(* Logix 5000 project; controller VFX vendor 1 type 14 code 177 rev 31.11; software revision 31.00 *)

TASK LazyTask (periodic, rate 10 ms, priority 10, watchdog 500 ms) : Operator_Interface
TASK MainTask (continuous, watchdog 500 ms) : MainProgram, fanucProgram, VFX
TASK SafetyTask (periodic, rate 20 ms, priority 10, watchdog 20 ms, safety) : SafetyProgram

MODULES
   Local : vendor 1 type 14 code 177 (Compact 0, rev 31.11)
      IPC : ETHERNET-MODULE (Ethernet 192.168.1.253, rev 1.1, Output RPI 10 ms)
      TURCK_4AI : vendor 48 type 12 code 14025 (Ethernet 192.168.1.20, rev 2.7, StandardDataDriven RPI 20 ms)
      fanuc : vendor 356 type 140 code 40 (Ethernet 192.168.1.41, rev 3.1, StandardDataDriven RPI 32 ms, A_Safety_Output RPI 20 ms, B_Safety_Input RPI 10 ms)
      pointIO : 1734-AENTR (Ethernet 192.168.1.21, rev 5.1, Output RPI 20 ms)
         di8 : 1734-IB8 (PointIO 3, rev 3.1)
         ai2 : 1734-IE2V (PointIO 5, rev 3.1, Input RPI 80 ms)
         do8 : 1734-OB8 (PointIO 4, rev 3.1)
         si8 : vendor 1 type 35 code 15 (PointIO 1, rev 2.1, Input RPI 10 ms, Output RPI 20 ms)
         so8 : vendor 1 type 35 code 16 (PointIO 2, rev 2.1, Input RPI 10 ms, Output RPI 20 ms)
END_MODULES

TYPE BOXTYPE :
STRUCT
   name : STRING;
   fiducial1 : POSREG_T;
   fiducial2 : POSREG_T;
   slot00 : POSREG_T;
   rowpitch : DINT;
   colpitch : DINT;
   numrows : DINT;
   numcols : DINT;
END_STRUCT
END_TYPE

TYPE Buttons :
STRUCT
   Start : BOOL;
   Stop : BOOL;
   FaultReset : BOOL;
   EStopReset : BOOL;
   Request : BOOL;
END_STRUCT
END_TYPE

TYPE FANUC_DIN1_T :   // FANUC I/O Structure
STRUCT
   dw0 : FANUC_DWORDI10_T;
   dw1 : FANUC_DWORDI11_T;
   dw2 : FANUC_DWORDI12_T;
   dw3 : FANUC_DWORDI13_T;
END_STRUCT
END_TYPE

TYPE FANUC_DIO :
STRUCT
   camera_trigger_req : BOOL;
   gripper_hasItem : BOOL;
   tool_engage_req : BOOL;
   tool_release_req : BOOL;
   gripper_open_req : BOOL;
   gripper_close_req : BOOL;
   laser_trigger_req : BOOL;
   mode_AUTO : BOOL;
   mode_ESTOP : BOOL;
   mode_T1 : BOOL;
   camera_trigger_ACK : BOOL;
   gripper_isOpen : BOOL;
   laser_trigger_ACK : BOOL;
   tool_isEngaged : BOOL;
   toolnest1_isOpen : BOOL;
   toolnest2_isOpen : BOOL;
   toolnest3_isOpen : BOOL;
   light : SINT;
   gripper_isClosed : BOOL;
END_STRUCT
END_TYPE

TYPE FANUC_DOUT1_T :   // FANUC I/O Structure
STRUCT
   dw0 : FANUC_DWORDO10_T;
   dw1 : FANUC_DWORDO11_T;
   dw2 : FANUC_DWORDO12_T;
   dw3 : FANUC_DWORDO13_T;
END_STRUCT
END_TYPE

TYPE FANUC_DWORDI10_T :   // FANUC I/O Structure
STRUCT
   Wago_analog_input_1_DI1_GI1_1 : BOOL;
   Wago_analog_input_1_DI2_GI1_2 : BOOL;
   Wago_analog_input_1_DI3_GI1_4 : BOOL;
   Wago_analog_input_1_DI4_GI1_8 : BOOL;
   Wago_analog_input_1_DI5_GI1_16 : BOOL;
   Wago_analog_input_1_DI6_GI1_32 : BOOL;
   Wago_analog_input_1_DI7_GI1_64 : BOOL;
   Wago_analog_input_1_DI8_GI1_128 : BOOL;
   Wago_analog_input_1_DI9_GI1_1 : BOOL;
   Wago_analog_input_1_DI10_GI1_2 : BOOL;
   Wago_analog_input_1_DI11_GI1_4 : BOOL;
   Wago_analog_input_1_DI12_GI1_8 : BOOL;
   Wago_analog_input_1_DI13_GI1_16 : BOOL;
   Wago_analog_input_1_DI14_GI1_32 : BOOL;
   Wago_analog_input_1_DI15_GI1_64 : BOOL;
   Wago_analog_input_1_DI16_GI1_128 : BOOL;
   Wago_analog_input_2_DI17_GI2_1 : BOOL;
   Wago_analog_input_2_DI18_GI2_2 : BOOL;
   Wago_analog_input_2_DI19_GI2_4 : BOOL;
   Wago_analog_input_2_DI20_GI2_8 : BOOL;
   Wago_analog_input_2_DI21_GI2_16 : BOOL;
   Wago_analog_input_2_DI22_GI2_32 : BOOL;
   Wago_analog_input_2_DI23_GI2_64 : BOOL;
   Wago_analog_input_2_DI24_GI2_128 : BOOL;
   Wago_analog_input_2_DI25_GI2_1 : BOOL;
   Wago_analog_input_2_DI26_GI2_2 : BOOL;
   Wago_analog_input_2_DI27_GI2_4 : BOOL;
   Wago_analog_input_2_DI28_GI2_8 : BOOL;
   Wago_analog_input_2_DI29_GI2_16 : BOOL;
   Wago_analog_input_2_DI30_GI2_32 : BOOL;
   Wago_analog_input_2_DI31_GI2_64 : BOOL;
   Wago_analog_input_2_DI32_GI2_128 : BOOL;
END_STRUCT
END_TYPE

TYPE FANUC_DWORDI11_T :   // FANUC I/O Structure
STRUCT
   DI33 : BOOL;
   DI34 : BOOL;
   DI35 : BOOL;
   DI36 : BOOL;
   DI37 : BOOL;
   DI38 : BOOL;
   DI39 : BOOL;
   DI40 : BOOL;
   DI41 : BOOL;
   DI42 : BOOL;
   DI43 : BOOL;
   DI44 : BOOL;
   DI45 : BOOL;
   DI46 : BOOL;
   DI47 : BOOL;
   DI48 : BOOL;
   DI49 : BOOL;
   DI50 : BOOL;
   DI51 : BOOL;
   DI52 : BOOL;
   DI53 : BOOL;
   DI54 : BOOL;
   DI55 : BOOL;
   DI56 : BOOL;
   DI57 : BOOL;
   DI58 : BOOL;
   DI59 : BOOL;
   DI60 : BOOL;
   DI61 : BOOL;
   DI62 : BOOL;
   DI63 : BOOL;
   DI64 : BOOL;
END_STRUCT
END_TYPE

TYPE FANUC_DWORDI12_T :   // FANUC I/O Structure
STRUCT
   IMSTP_DI65_UI1 : BOOL;
   Hold_DI66_UI2 : BOOL;
   SFSPD_DI67_UI3 : BOOL;
   Cycle_stop_DI68_UI4 : BOOL;
   Fault_reset_DI69_UI5 : BOOL;
   Start_DI70_UI6 : BOOL;
   Home_DI71_UI7 : BOOL;
   Enable_DI72_UI8 : BOOL;
   RSR1PNS1STYLE1_DI73_UI9 : BOOL;
   RSR2PNS2STYLE2_DI74_UI10 : BOOL;
   RSR3PNS3STYLE3_DI75_UI11 : BOOL;
   RSR4PNS4STYLE4_DI76_UI12 : BOOL;
   RSR5PNS5STYLE5_DI77_UI13 : BOOL;
   RSR6PNS6STYLE6_DI78_UI14 : BOOL;
   RSR7PNS7STYLE7_DI79_UI15 : BOOL;
   RSR8PNS8STYLE8_DI80_UI16 : BOOL;
   PNS_strobe_DI81_UI17 : BOOL;
   Prod_start_DI82_UI18 : BOOL;
   DI83 : BOOL;
   DI84 : BOOL;
   DI85 : BOOL;
   DI86 : BOOL;
   DI87 : BOOL;
   DI88 : BOOL;
   DI89 : BOOL;
   DI90 : BOOL;
   DI91 : BOOL;
   DI92 : BOOL;
   DI93 : BOOL;
   DI94 : BOOL;
   DI95 : BOOL;
   DI96 : BOOL;
END_STRUCT
END_TYPE

TYPE FANUC_DWORDI13_T :   // FANUC I/O Structure
STRUCT
   DI97 : BOOL;
   DI98 : BOOL;
   DI99 : BOOL;
   Cognex_trig_ready_DI100 : BOOL;
   Cognex_trig_ack_DI101 : BOOL;
   Cognex_acquiring_DI102 : BOOL;
   Cognex_missed_ack_DI103 : BOOL;
   Cognex_online_DI104 : BOOL;
   Cognex_inspecting_DI105 : BOOL;
   Cognex_inspect_complete_DI106 : BOOL;
   Cognex_buffer_overrun_DI107 : BOOL;
   Cognex_results_valid_DI108 : BOOL;
   Cognex_job_loading_DI109 : BOOL;
   Cognex_job_load_complete_DI110 : BOOL;
   Cognex_job_load_failed_DI111 : BOOL;
   Cognex_exposure_complete_DI112 : BOOL;
   Cognex_job_pass_DI113 : BOOL;
   DI114 : BOOL;
   DI115 : BOOL;
   DI116 : BOOL;
   DI117 : BOOL;
   DI118 : BOOL;
   DI119 : BOOL;
   DI120 : BOOL;
   DI121 : BOOL;
   DI122 : BOOL;
   DI123 : BOOL;
   DI124 : BOOL;
   DI125 : BOOL;
   DI126 : BOOL;
   DI127 : BOOL;
   DI128 : BOOL;
END_STRUCT
END_TYPE

TYPE FANUC_DWORDO10_T :   // FANUC I/O Structure
STRUCT
   Camera_Trigger_DO1 : BOOL;
   Camera_Continouts_DO2 : BOOL;
   Laser_Trigger_DO3 : BOOL;
   Laser_Continous_DO4 : BOOL;
   DO5 : BOOL;
   DO6 : BOOL;
   DO7 : BOOL;
   DO8 : BOOL;
   DO9 : BOOL;
   DO10 : BOOL;
   DO11 : BOOL;
   DO12 : BOOL;
   DO13 : BOOL;
   DO14 : BOOL;
   DO15 : BOOL;
   DO16 : BOOL;
   DO17 : BOOL;
   DO18 : BOOL;
   DO19 : BOOL;
   DO20 : BOOL;
   DO21 : BOOL;
   DO22 : BOOL;
   DO23 : BOOL;
   DO24 : BOOL;
   DO25 : BOOL;
   DO26 : BOOL;
   DO27 : BOOL;
   DO28 : BOOL;
   DO29 : BOOL;
   DO30 : BOOL;
   DO31 : BOOL;
   DO32 : BOOL;
END_STRUCT
END_TYPE

TYPE FANUC_DWORDO11_T :   // FANUC I/O Structure
STRUCT
   DO33 : BOOL;
   DO34 : BOOL;
   DO35 : BOOL;
   DO36 : BOOL;
   DO37 : BOOL;
   DO38 : BOOL;
   DO39 : BOOL;
   DO40 : BOOL;
   DO41 : BOOL;
   DO42 : BOOL;
   DO43 : BOOL;
   DO44 : BOOL;
   DO45 : BOOL;
   DO46 : BOOL;
   DO47 : BOOL;
   DO48 : BOOL;
   DO49 : BOOL;
   DO50 : BOOL;
   DO51 : BOOL;
   DO52 : BOOL;
   DO53 : BOOL;
   DO54 : BOOL;
   DO55 : BOOL;
   DO56 : BOOL;
   DO57 : BOOL;
   DO58 : BOOL;
   DO59 : BOOL;
   DO60 : BOOL;
   DO61 : BOOL;
   DO62 : BOOL;
   DO63 : BOOL;
   DO64 : BOOL;
END_STRUCT
END_TYPE

TYPE FANUC_DWORDO12_T :   // FANUC I/O Structure
STRUCT
   Cmd_enabled_DO65_UO1 : BOOL;
   System_ready_DO66_UO2 : BOOL;
   Prg_running_DO67_UO3 : BOOL;
   Prg_paused_DO68_UO4 : BOOL;
   Motion_held_DO69_UO5 : BOOL;
   Fault_DO70_UO6 : BOOL;
   At_perch_DO71_UO7 : BOOL;
   TP_enabled_DO72_UO8 : BOOL;
   Batt_alarm_DO73_UO9 : BOOL;
   Busy_DO74_UO10 : BOOL;
   ACK1SNO1_DO75_UO11 : BOOL;
   ACK2SNO2_DO76_UO12 : BOOL;
   ACK3SNO3_DO77_UO13 : BOOL;
   ACK4SNO4_DO78_UO14 : BOOL;
   ACK5SNO5_DO79_UO15 : BOOL;
   ACK6SNO6_DO80_UO16 : BOOL;
   ACK7SNO7_DO81_UO17 : BOOL;
   ACK8SNO8_DO82_UO18 : BOOL;
   SNACK_DO83_UO19 : BOOL;
   Reserved_DO84_UO20 : BOOL;
   DO85 : BOOL;
   DO86 : BOOL;
   DO87 : BOOL;
   DO88 : BOOL;
   DO89 : BOOL;
   DO90 : BOOL;
   DO91 : BOOL;
   DO92 : BOOL;
   DO93 : BOOL;
   DO94 : BOOL;
   DO95 : BOOL;
   DO96 : BOOL;
END_STRUCT
END_TYPE

TYPE FANUC_DWORDO13_T :   // FANUC I/O Structure
STRUCT
   DO97 : BOOL;
   DO98 : BOOL;
   DO99 : BOOL;
   Cognex_trigger_enable_DO100 : BOOL;
   Cognex_trigger_DO101 : BOOL;
   Cognex_buffer_results_en_DO102 : BOOL;
   Cognex_inspect_result_ok_DO103 : BOOL;
   Cognex_reserved_DO104 : BOOL;
   Cognex_reserved_DO105 : BOOL;
   Cognex_reserved_DO106 : BOOL;
   Cognex_set_offline_DO107 : BOOL;
   Cognex_soft_event_0_DO108 : BOOL;
   Cognex_soft_event_1_DO109 : BOOL;
   Cognex_soft_event_2_DO110 : BOOL;
   Cognex_soft_event_3_DO111 : BOOL;
   Cognex_soft_event_4_DO112 : BOOL;
   Cognex_soft_event_5_DO113 : BOOL;
   Cognex_soft_event_6_DO114 : BOOL;
   Cognex_soft_event_7_DO115 : BOOL;
   Cognex_reserved_DO116 : BOOL;
   Cognex_reserved_DO117 : BOOL;
   Cognex_reserved_DO118 : BOOL;
   Cognex_reserved_DO119 : BOOL;
   Cognex_reserved_DO120 : BOOL;
   Cognex_reserved_DO121 : BOOL;
   Cognex_reserved_DO122 : BOOL;
   Cognex_reserved_DO123 : BOOL;
   Cognex_reserved_DO124 : BOOL;
   Cognex_reserved_DO125 : BOOL;
   Cognex_reserved_DO126 : BOOL;
   Cognex_reserved_DO127 : BOOL;
   Cognex_reserved_DO128 : BOOL;
END_STRUCT
END_TYPE

TYPE FANUC_EDA_T :
STRUCT
   out : FANUC_I_T;
   in : FANUC_O_T;
END_STRUCT
END_TYPE

TYPE FANUC_I_T :
STRUCT
   dout : FANUC_DIN1_T;
   speed_max_R1 : DINT;
   speed_camera_R2 : DINT;
   speed_laser_R3 : DINT;
   speed_approach_R4 : DINT;
   R5 : DINT;
   R6 : DINT;
   R7 : DINT;
   R8 : DINT;
   speedj_max_R9 : DINT;
   speedj_payload_R10 : DINT;
   boxtype_numrows_R11 : DINT;
   boxtype_numcols_R12 : DINT;
   camera_getmode_R13 : DINT;
   laser_distance_R14 : DINT;
   camera_getfiducl_R15 : DINT;
   skip_perch_R16 : DINT;
   R17 : DINT;
   boxtype_ID_R18 : DINT;
   boxtype_rowpitch_R19 : DINT;
   boxtype_colpitch_R20 : DINT;
   target_boxnum_R21 : DINT;
   target_slotrow_R22 : DINT;
   target_slotcol_R23 : DINT;
   R24 : DINT;
   boxtype_fid1_PR1_G1 : POSREG_T;
   boxtype_fid2_PR2_G1 : POSREG_T;
   boxtype_slot00_PR3_G1 : POSREG_T;
   boxframe_offset_PR4_G1 : POSREG_T;
END_STRUCT
END_TYPE

TYPE FANUC_MASTER :
STRUCT
   uop : FANUC_UOPS;
   reg : FANUC_REGISTERS;
   dio : FANUC_DIO;
END_STRUCT
END_TYPE

TYPE FANUC_O_T :
STRUCT
   din : FANUC_DOUT1_T;
   speed_max_R1 : DINT;
   speed_camera_R2 : DINT;
   speed_laser_R3 : DINT;
   speed_approach_R4 : DINT;
   R5 : DINT;
   R6 : DINT;
   R7 : DINT;
   R8 : DINT;
   speedj_max_R9 : DINT;
   speedj_payload_R10 : DINT;
   boxtype_numrows_R11 : DINT;
   boxtype_numcols_R12 : DINT;
   camera_getmode_R13 : DINT;
   laser_distance_R14 : DINT;
   camera_getfiducl_R15 : DINT;
   skip_perch_R16 : DINT;
   R17 : DINT;
   boxtype_ID_R18 : DINT;
   boxtype_rowpitch_R19 : DINT;
   boxtype_colpitch_R20 : DINT;
   target_boxnum_R21 : DINT;
   target_slotrow_R22 : DINT;
   target_slotcol_R23 : DINT;
   R24 : DINT;
   R25 : DINT;
   R26 : DINT;
   R27 : DINT;
   R28 : DINT;
   R29 : DINT;
   R30 : DINT;
   style_result_R31 : DINT;
   row_current_R32 : DINT;
   boxtype_fid1_PR1_G1 : POSREG_T;
   boxtype_fid2_PR2_G1 : POSREG_T;
   boxtype_slot00_PR3_G1 : POSREG_T;
   boxframe_offset_PR4_G1 : POSREG_T;
   eda1_PR5_G1 : POSREG_T;
   eda2_PR6_G1 : POSREG_T;
   CURPOS_G1 : POSREG_T;
END_STRUCT
END_TYPE

TYPE FANUC_REGISTERS :
STRUCT
   boxframe_offset : POSREG_T;
   boxframe_offset_ACK : POSREG_T;
   boxtype : BOXTYPE;
   boxtype_ACK : BOXTYPE;
   laser_distance : DINT;
   speed_approach : DINT;
   speed_max : DINT;
   speed_payload : DINT;
   speed_toolchange : DINT;
   target_boxnum : DINT;
   target_slotrow : DINT;
   target_slotcol : DINT;
   target_tool_ID : DINT;
   CURPOS : POSREG_T;
   EDA1 : POSREG_T;
   EDA2 : POSREG_T;
   laser_distance_ACK : DINT;
   speed_approach_ACK : DINT;
   speed_max_ACK : DINT;
   speed_payload_ACK : DINT;
   speed_toolchange_ACK : DINT;
   speedj_max_ACK : DINT;
   speedJ_payload_ACK : DINT;
   target_boxnum_ACK : DINT;
   target_slotrow_ACK : DINT;
   target_slotcol_ACK : DINT;
   current_tool_ID : DINT;
   target_fiducial : DINT;
   target_fiducial_ACK : DINT;
   style_result : DINT;
END_STRUCT
END_TYPE

TYPE FANUC_UOPS :
STRUCT
   cycle_stop : BOOL;
   enable : BOOL;
   fault_reset : BOOL;
   hold : BOOL;
   home : BOOL;
   IMSTP : BOOL;
   pns_strobe : BOOL;
   prod_start : BOOL;
   style : SINT;
   SFSPD : BOOL;
   start : BOOL;
   style_ACK : SINT;
   at_perch : BOOL;
   batt_alarm : BOOL;
   busy : BOOL;
   cmd_enabled : BOOL;
   fault : BOOL;
   motion_held : BOOL;
   prg_paused : BOOL;
   prg_running : BOOL;
   reserved : BOOL;
   SNACK : BOOL;
   system_ready : BOOL;
   TP_enabled : BOOL;
END_STRUCT
END_TYPE

TYPE Pedestal_Lights :
STRUCT
   Start : BOOL;
   Stop : BOOL;
   FaultReset : BOOL;
   EStopReset : BOOL;
   Request : BOOL;
   EStop : BOOL;
   White : BOOL;
   Blue : BOOL;
   Green : BOOL;
   Amber : BOOL;
   Red : BOOL;
   White_Flasher : BOOL;
   Blue_Flasher : BOOL;
   Green_Flasher : BOOL;
   Amber_Flasher : BOOL;
   Red_Flasher : BOOL;
END_STRUCT
END_TYPE

TYPE POSREG_T :   // FANUC Position Register (Cartesian Mode)
STRUCT
   uframe : INT;
   utool : INT;
   X : REAL;
   Y : REAL;
   Z : REAL;
   W : REAL;
   P : REAL;
   R : REAL;
   turn1 : SINT;
   turn2 : SINT;
   turn3 : SINT;
   front : BOOL;
   up : BOOL;
   left : BOOL;
   flip : BOOL;
   ext : REAL[3];
END_STRUCT
END_TYPE

VAR_GLOBAL   (* controller tags *)
   boxtypes : BOXTYPE[10] := ([0].name := 'tote', [0].fiducial1.uframe := -1, [0].fiducial1.front := 1, [0].fiducial1.up := 1, [0].fiducial1.left := 1, [0].fiducial2.uframe := -1, [0].fiducial2.X := 580.0, [0].fiducial2.Z := -220.0, [0].fiducial2.front := 1, [0].fiducial2.up := 1, [0].fiducial2.left := 1, [0].slot00.uframe := -1, [0].slot00.X := 60.0, [0].slot00.Y := 60.0, [0].slot00.Z := -295.0, [0].slot00.front := 1, [0].slot00.up := 1, [0].slot00.left := 1, [0].rowpitch := 42164, [0].colpitch := 128016, [0].numrows := 12, [0].numcols := 2, [1].name := 'carton1', [1].fiducial1.uframe := 63, [1].fiducial1.utool := 31, [1].fiducial1.X := 100.0, [1].fiducial1.Y := 40.0, [1].fiducial1.front := 1, [1].fiducial1.up := 1, [1].fiducial1.left := 1, [1].fiducial2.uframe := 63, [1].fiducial2.utool := 31, [1].fiducial2.X := 377.0, [1].fiducial2.Z := -220.0, [1].fiducial2.front := 1, [1].fiducial2.up := 1, [1].fiducial2.left := 1, [1].slot00.uframe := -1, [1].slot00.X := -18.5, [1].slot00.Y := 60.0, [1].slot00.Z := -295.0, [1].slot00.front := 1, [1].slot00.up := 1, [1].slot00.left := 1, [1].rowpitch := 47350, [1].colpitch := 122428, [1].numrows := 10, [1].numcols := 2);
   fanuc : FANUC_MASTER := (uop.enable := 1, uop.hold := 1, uop.IMSTP := 1, uop.style := 3, uop.SFSPD := 1, uop.cmd_enabled := 1, reg.boxframe_offset.uframe := -1, reg.boxframe_offset.X := 11.01, reg.boxframe_offset.Y := -9.029, reg.boxtype.name := 'tote', reg.boxtype.fiducial1.uframe := -1, reg.boxtype.fiducial1.front := 1, reg.boxtype.fiducial1.up := 1, reg.boxtype.fiducial1.left := 1, reg.boxtype.fiducial2.uframe := -1, reg.boxtype.fiducial2.X := 580.0, reg.boxtype.fiducial2.Z := -220.0, reg.boxtype.fiducial2.front := 1, reg.boxtype.fiducial2.up := 1, reg.boxtype.fiducial2.left := 1, reg.boxtype.slot00.uframe := -1, reg.boxtype.slot00.X := 60.0, reg.boxtype.slot00.Y := 60.0, reg.boxtype.slot00.Z := -295.0, reg.boxtype.slot00.front := 1, reg.boxtype.slot00.up := 1, reg.boxtype.slot00.left := 1, reg.boxtype.rowpitch := 42164, reg.boxtype.colpitch := 128016, reg.boxtype.numrows := 12, reg.boxtype.numcols := 2, reg.speed_approach := 1000, reg.speed_max := 2000, reg.speed_payload := 2000, reg.speed_toolchange := 2000, reg.target_boxnum := 7, reg.target_slotrow := 11, reg.target_slotcol := 1, reg.CURPOS.uframe := 7, reg.CURPOS.utool := 1, reg.CURPOS.X := 523.80383, reg.CURPOS.Y := -68.01611, reg.CURPOS.Z := -294.99994, reg.CURPOS.W := -1.6060338e-05, reg.CURPOS.P := 0.00042976913, reg.CURPOS.R := 1.6143189e-05, reg.CURPOS.front := 1, reg.CURPOS.up := 1, reg.EDA1.uframe := 255, reg.EDA1.utool := 255, reg.EDA1.X := nan, reg.EDA1.Y := nan, reg.EDA1.Z := nan, reg.EDA1.W := nan, reg.EDA1.P := nan, reg.EDA1.R := nan, reg.style_result := 1);
   fanuc_auto_enable : BOOL := 1;
   Fanuc_AUTO_OFF : BOOL := 1;
   Fanuc_ESTOP : EMERGENCY_STOP := (ChannelA := 1, ChannelB := 1, CircuitReset := 1, FaultReset := 1, O1 := 1);
   Fanuc_ESTOP_IN : BOOL := 1;
   Fanuc_ESTOP_OUT : BOOL := 1;
   Fanuc_FENCE : BOOL := 1;
   fanuc_IPC_start : BOOL;
   fanuc_permissive : BOOL := 1;
   fanuc_run : BOOL := 1;
   fanuc_s1 : FANUC_EDA_T := (out.dout.dw2.IMSTP_DI65_UI1 := 1, out.dout.dw2.Hold_DI66_UI2 := 1, out.dout.dw2.SFSPD_DI67_UI3 := 1, out.dout.dw2.Enable_DI72_UI8 := 1, out.dout.dw2.RSR1PNS1STYLE1_DI73_UI9 := 1, out.dout.dw2.RSR2PNS2STYLE2_DI74_UI10 := 1, out.speed_max_R1 := 2000, out.speed_camera_R2 := 2000, out.speed_laser_R3 := 1000, out.speed_approach_R4 := 2000, out.speedj_max_R9 := 100, out.speedj_payload_R10 := 100, out.boxtype_numrows_R11 := 12, out.boxtype_numcols_R12 := 2, out.boxtype_rowpitch_R19 := 42164, out.boxtype_colpitch_R20 := 128016, out.target_boxnum_R21 := 7, out.target_slotrow_R22 := 11, out.target_slotcol_R23 := 1, out.boxtype_fid1_PR1_G1.uframe := -1, out.boxtype_fid1_PR1_G1.front := 1, out.boxtype_fid1_PR1_G1.up := 1, out.boxtype_fid1_PR1_G1.left := 1, out.boxtype_fid2_PR2_G1.uframe := -1, out.boxtype_fid2_PR2_G1.X := 580.0, out.boxtype_fid2_PR2_G1.Z := -220.0, out.boxtype_fid2_PR2_G1.front := 1, out.boxtype_fid2_PR2_G1.up := 1, out.boxtype_fid2_PR2_G1.left := 1, out.boxtype_slot00_PR3_G1.uframe := -1, out.boxtype_slot00_PR3_G1.X := 60.0, out.boxtype_slot00_PR3_G1.Y := 60.0, out.boxtype_slot00_PR3_G1.Z := -295.0, out.boxtype_slot00_PR3_G1.front := 1, out.boxtype_slot00_PR3_G1.up := 1, out.boxtype_slot00_PR3_G1.left := 1, out.boxframe_offset_PR4_G1.uframe := -1, out.boxframe_offset_PR4_G1.X := 11.01, out.boxframe_offset_PR4_G1.Y := -9.029, in.din.dw2.Cmd_enabled_DO65_UO1 := 1, in.din.dw2.System_ready_DO66_UO2 := 1, in.speed_max_R1 := 2000, in.speed_camera_R2 := 2000, in.speed_laser_R3 := 1000, in.speed_approach_R4 := 2000, in.speedj_max_R9 := 100, in.speedj_payload_R10 := 100, in.boxtype_numrows_R11 := 12, in.boxtype_numcols_R12 := 2, in.boxtype_rowpitch_R19 := 42164, in.boxtype_colpitch_R20 := 128016, in.target_boxnum_R21 := 7, in.target_slotrow_R22 := 11, in.target_slotcol_R23 := 1, in.style_result_R31 := 1, in.boxtype_fid1_PR1_G1.uframe := 255, in.boxtype_fid1_PR1_G1.utool := 255, in.boxtype_fid1_PR1_G1.front := 1, in.boxtype_fid1_PR1_G1.up := 1, in.boxtype_fid1_PR1_G1.left := 1,
        in.boxtype_fid2_PR2_G1.uframe := 255, in.boxtype_fid2_PR2_G1.utool := 255, in.boxtype_fid2_PR2_G1.X := 580.0, in.boxtype_fid2_PR2_G1.Z := -220.0, in.boxtype_fid2_PR2_G1.front := 1, in.boxtype_fid2_PR2_G1.up := 1, in.boxtype_fid2_PR2_G1.left := 1, in.boxtype_slot00_PR3_G1.uframe := 255, in.boxtype_slot00_PR3_G1.utool := 255, in.boxtype_slot00_PR3_G1.X := 60.0, in.boxtype_slot00_PR3_G1.Y := 60.0, in.boxtype_slot00_PR3_G1.Z := -295.0, in.boxtype_slot00_PR3_G1.front := 1, in.boxtype_slot00_PR3_G1.up := 1, in.boxtype_slot00_PR3_G1.left := 1, in.boxframe_offset_PR4_G1.uframe := 255, in.boxframe_offset_PR4_G1.utool := 255, in.boxframe_offset_PR4_G1.X := 11.01, in.boxframe_offset_PR4_G1.Y := -9.029, in.eda1_PR5_G1.uframe := 255, in.eda1_PR5_G1.utool := 255, in.eda1_PR5_G1.X := nan, in.eda1_PR5_G1.Y := nan, in.eda1_PR5_G1.Z := nan, in.eda1_PR5_G1.W := nan, in.eda1_PR5_G1.P := nan, in.eda1_PR5_G1.R := nan, in.eda2_PR6_G1.uframe := 255, in.eda2_PR6_G1.utool := 255, in.eda2_PR6_G1.X := nan, in.eda2_PR6_G1.Y := nan, in.eda2_PR6_G1.Z := nan, in.eda2_PR6_G1.W := nan, in.eda2_PR6_G1.P := nan, in.eda2_PR6_G1.R := nan, in.CURPOS_G1.uframe := 7, in.CURPOS_G1.utool := 1, in.CURPOS_G1.X := 523.80383, in.CURPOS_G1.Y := -68.01611, in.CURPOS_G1.Z := -294.99994, in.CURPOS_G1.W := -1.6060338e-05, in.CURPOS_G1.P := 0.00042976913, in.CURPOS_G1.R := 1.6143189e-05, in.CURPOS_G1.front := 1, in.CURPOS_G1.up := 1);
   fanuc_style_start : BOOL;
   fanuc_target_boxtype : DINT;
   fanuc_target_valid : BOOL := 1;
   FENCE_CLOSED : BOOL := 1;
   HMI_Buttons : Buttons;
   HMI_Buttons2 : BOOL;
   HMI_ESTOP_Reset : BOOL;
   light_flasher : TIMER := (PRE := 500, ACC := 500, EN := 1, DN := 1);
   light_flasher2 : TIMER := (PRE := 500, ACC := 220, EN := 1, TT := 1);
   out_fail2 : BOOL := 1;
   out_pass2 : BOOL;
   output_pulse2 : DINT := 250;
   Panel_HMI_Lights : Pedestal_Lights;
   Panel_Stack_Amber : BOOL;
   Panel_Stack_Amber_Flasher : BOOL;
   Panel_Stack_Green : BOOL;
   Panel_Stack_Green_Flasher : BOOL := 1;
   Panel_Stack_Red : BOOL;
   Panel_Stack_Red_Flasher : BOOL;
   Pedestal1_ESTOP : EMERGENCY_STOP := (ResetType := 1, ChannelA := 1, ChannelB := 1, CircuitReset := 1, O1 := 1);
   Pedestal2_ESTOP : EMERGENCY_STOP := (ResetType := 1, ChannelA := 1, ChannelB := 1, CircuitReset := 1, O1 := 1);
   Safety_EStopReset : BOOL := 1;
   Safety_FaultReset : BOOL := 1;
   shhhhhhhhhh : BOOL;
   step_robot_command : DINT := 40;
   System_ESTOP : BOOL := 1;
   System_EStopReset : BOOL := 1;
   System_EStopResetReq : BOOL;
   System_FaultReset2 : BOOL;
   system_running : BOOL;
   system_running_debounce : TIMER := (PRE := 500, ACC := 500);
   System_Start : BOOL;
   System_Start2 : BOOL;
   System_Stop : BOOL;
   System_Stop2 : BOOL;
   tmr_pulse_fanuc : TIMER := (PRE := 500);
   tmr_pulse_fanuc_done : TIMER := (PRE := 500);
   tmr_start_fanuc : TIMER := (PRE := 100);
   vfx_laser_distance : INT[2];
END_VAR

PROGRAM fanucProgram   (* main routine fanucRoutine *)

ROUTINE fanucRoutine   (* ladder *)
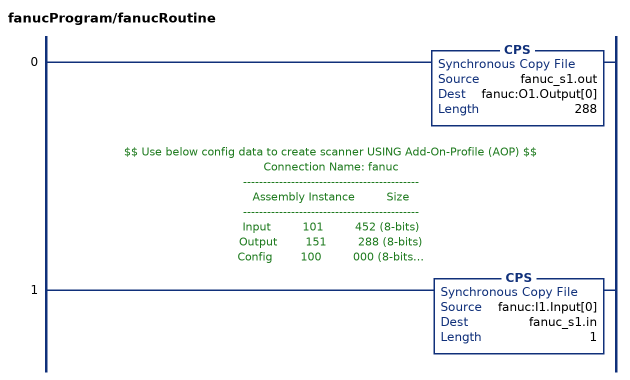
   0: CPS(fanuc_s1.out,fanuc:O1.Output[0],288);
   // $$ Use below config data to create scanner USING Add-On-Profile (AOP) $$
   //                   Connection Name: fanuc
   //                 --------------------------------------------
   //                   Assembly Instance         Size
   //                 --------------------------------------------
   //                   Input         101         452 (8-bits)
   //                   Output        151         288 (8-bits)
   //                   Config        100         000 (8-bits)
   //                 --------------------------------------------
   1: CPS(fanuc:I1.Input[0],fanuc_s1.in,1);
END_ROUTINE
END_PROGRAM

PROGRAM MainProgram   (* main routine MainRoutine *)

ROUTINE MainRoutine   (* ladder *)
   0 (stored rung type 13): ;
END_ROUTINE
END_PROGRAM

PROGRAM Operator_Interface   (* main routine Main_OI *)

ROUTINE Buttons_IO   (* ladder *)
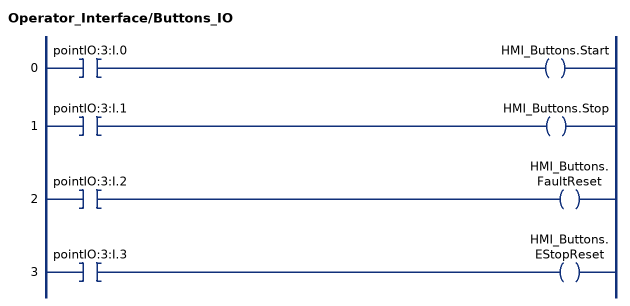
   0: XIC(pointIO:3:I.0)OTE(HMI_Buttons.Start);
   1: XIC(pointIO:3:I.1)OTE(HMI_Buttons.Stop);
   2: XIC(pointIO:3:I.2)OTE(HMI_Buttons.FaultReset);
   3: XIC(pointIO:3:I.3)OTE(HMI_Buttons.EStopReset);
END_ROUTINE

ROUTINE Buttons_Logic   (* ladder *)
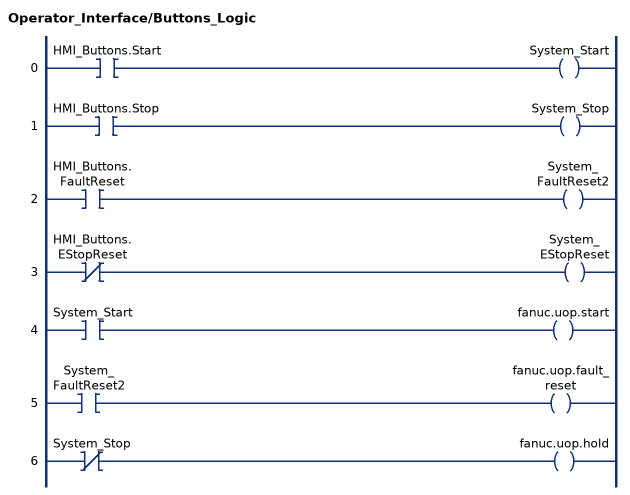
   0: XIC(HMI_Buttons.Start)OTE(System_Start);
   1: XIC(HMI_Buttons.Stop)OTE(System_Stop);
   2: XIC(HMI_Buttons.FaultReset)OTE(System_FaultReset2);
   3: XIO(HMI_Buttons.EStopReset)OTE(System_EStopReset);
   4: XIC(System_Start)OTE(fanuc.uop.start);
   5: XIC(System_FaultReset2)OTE(fanuc.uop.fault_reset);
   6: XIO(System_Stop)OTE(fanuc.uop.hold);
END_ROUTINE

ROUTINE Lights_IO   (* ladder *)
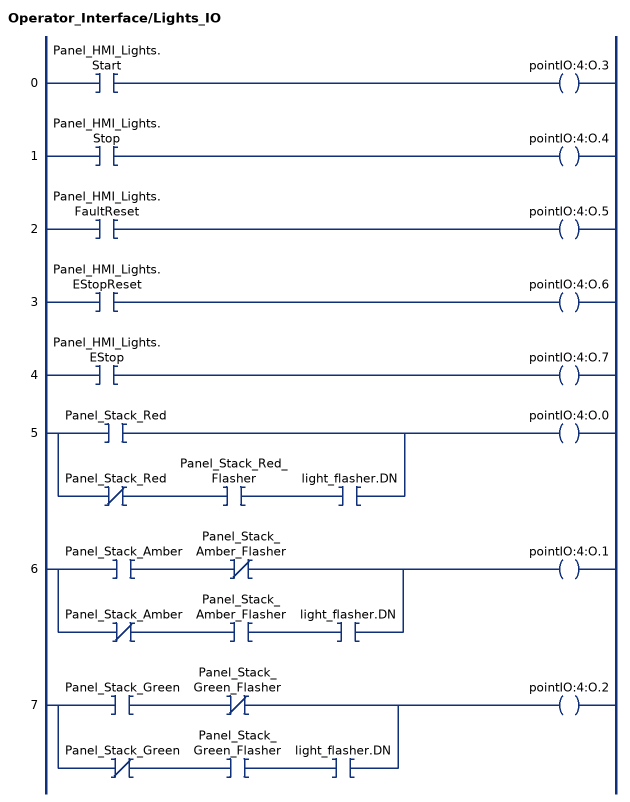
   0: XIC(Panel_HMI_Lights.Start)OTE(pointIO:4:O.3);
   1: XIC(Panel_HMI_Lights.Stop)OTE(pointIO:4:O.4);
   2: XIC(Panel_HMI_Lights.FaultReset)OTE(pointIO:4:O.5);
   3: XIC(Panel_HMI_Lights.EStopReset)OTE(pointIO:4:O.6);
   4: XIC(Panel_HMI_Lights.EStop)OTE(pointIO:4:O.7);
   5: [XIC(Panel_Stack_Red) ,XIO(Panel_Stack_Red) XIC(Panel_Stack_Red_Flasher) XIC(light_flasher.DN) ]OTE(pointIO:4:O.0);
   6: [XIC(Panel_Stack_Amber) XIO(Panel_Stack_Amber_Flasher) ,XIO(Panel_Stack_Amber) XIC(Panel_Stack_Amber_Flasher) XIC(light_flasher.DN) ]OTE(pointIO:4:O.1);
   7: [XIC(Panel_Stack_Green) XIO(Panel_Stack_Green_Flasher) ,XIO(Panel_Stack_Green) XIC(Panel_Stack_Green_Flasher) XIC(light_flasher.DN) ]OTE(pointIO:4:O.2);
END_ROUTINE

ROUTINE Lights_Logic   (* ladder *)
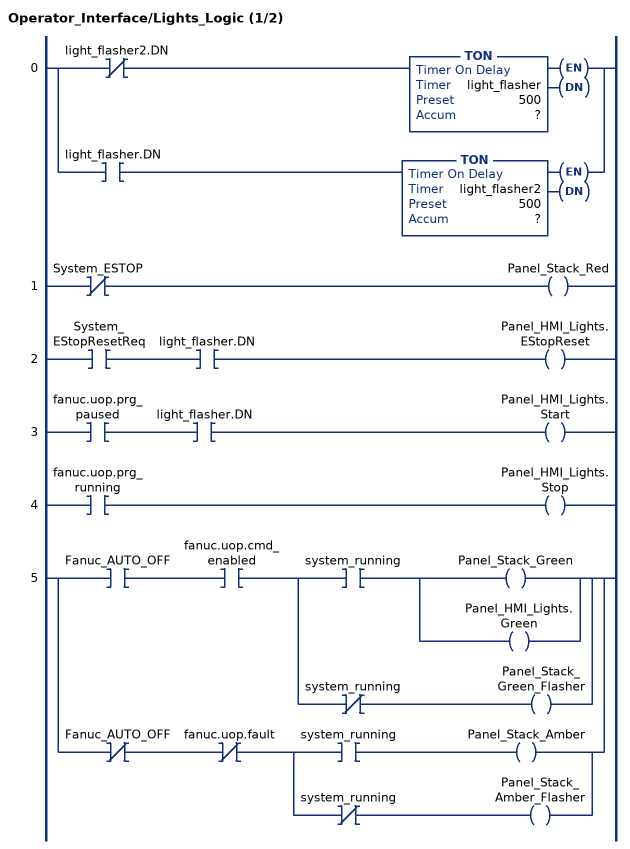
   0: [XIO(light_flasher2.DN) TON(light_flasher,?,?) ,XIC(light_flasher.DN) TON(light_flasher2,?,?) ];
   1: XIO(System_ESTOP)OTE(Panel_Stack_Red);
   2: XIC(System_EStopResetReq)XIC(light_flasher.DN)OTE(Panel_HMI_Lights.EStopReset);
   3: XIC(fanuc.uop.prg_paused)XIC(light_flasher.DN)OTE(Panel_HMI_Lights.Start);
   4: XIC(fanuc.uop.prg_running)OTE(Panel_HMI_Lights.Stop);
   5: [XIC(Fanuc_AUTO_OFF) XIC(fanuc.uop.cmd_enabled) [XIC(system_running) [OTE(Panel_Stack_Green) ,OTE(Panel_HMI_Lights.Green) ] ,XIO(system_running) OTE(Panel_Stack_Green_Flasher) ] ,XIO(Fanuc_AUTO_OFF) XIO(fanuc.uop.fault) [XIC(system_running) OTE(Panel_Stack_Amber) ,XIO(system_running) OTE(Panel_Stack_Amber_Flasher) ] ];
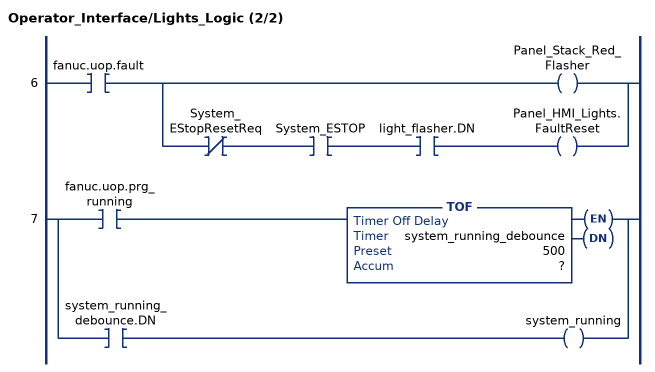
   6: XIC(fanuc.uop.fault)[OTE(Panel_Stack_Red_Flasher) ,XIO(System_EStopResetReq) XIC(System_ESTOP) XIC(light_flasher.DN) OTE(Panel_HMI_Lights.FaultReset) ];
   7: [XIC(fanuc.uop.prg_running) TOF(system_running_debounce,?,?) ,XIC(system_running_debounce.DN) OTE(system_running) ];
END_ROUTINE

ROUTINE Main_OI   (* ladder *)
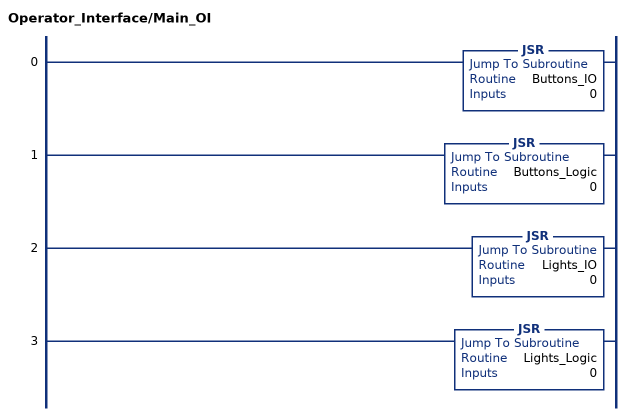
   0: JSR(Buttons_IO,0);
   1: JSR(Buttons_Logic,0);
   2: JSR(Lights_IO,0);
   3: JSR(Lights_Logic,0);
END_ROUTINE
END_PROGRAM

PROGRAM SafetyProgram   (* main routine MainRoutine, safety *)

ROUTINE ESTOPS   (* ladder *)
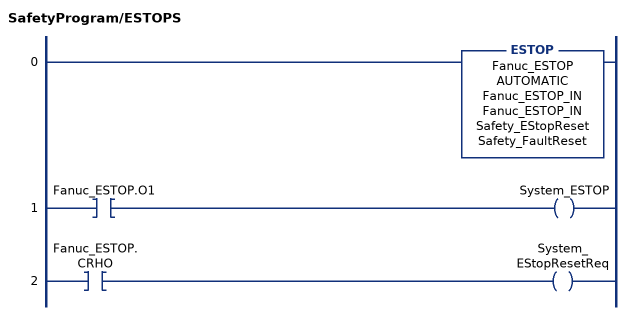
   0: ESTOP(Fanuc_ESTOP,AUTOMATIC,Fanuc_ESTOP_IN,Fanuc_ESTOP_IN,Safety_EStopReset,Safety_FaultReset);
   1: XIC(Fanuc_ESTOP.O1)OTE(System_ESTOP);
   2: XIC(Fanuc_ESTOP.CRHO)OTE(System_EStopResetReq);
END_ROUTINE

ROUTINE IO_Map   (* ladder *)
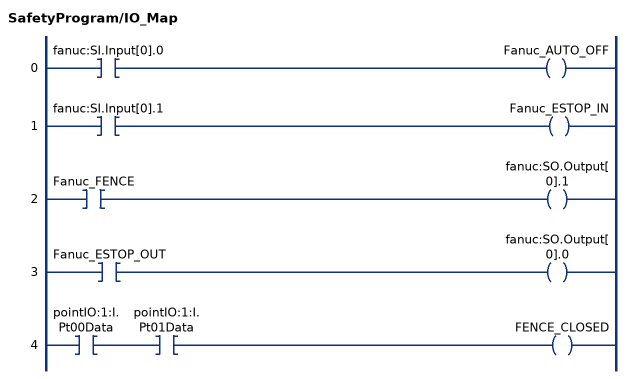
   0: XIC(fanuc:SI.Input[0].0)OTE(Fanuc_AUTO_OFF);
   1: XIC(fanuc:SI.Input[0].1)OTE(Fanuc_ESTOP_IN);
   2: XIC(Fanuc_FENCE)OTE(fanuc:SO.Output[0].1);
   3: XIC(Fanuc_ESTOP_OUT)OTE(fanuc:SO.Output[0].0);
   4: XIC(pointIO:1:I.Pt00Data)XIC(pointIO:1:I.Pt01Data)OTE(FENCE_CLOSED);
END_ROUTINE

ROUTINE MainRoutine   (* ladder *)
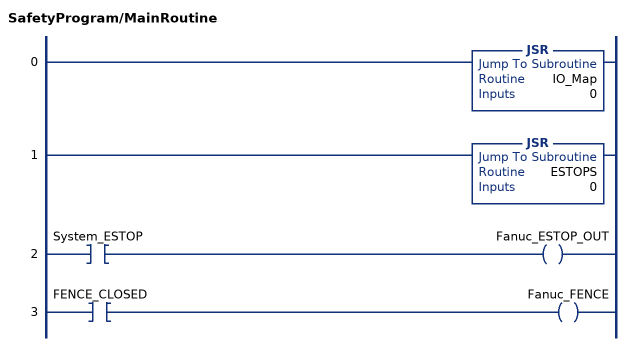
   0: JSR(IO_Map,0);
   1: JSR(ESTOPS,0);
   2: XIC(System_ESTOP)OTE(Fanuc_ESTOP_OUT);
   3: XIC(FENCE_CLOSED)OTE(Fanuc_FENCE);
END_ROUTINE
END_PROGRAM

PROGRAM VFX   (* main routine MainRoutine *)

ROUTINE Demo3   (* ladder *)
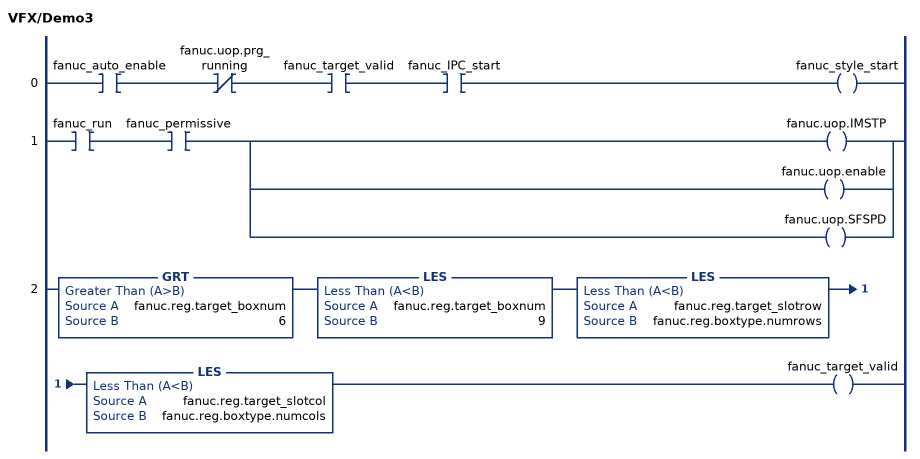
   0: XIC(fanuc_auto_enable)XIO(fanuc.uop.prg_running)XIC(fanuc_target_valid)XIC(fanuc_IPC_start)OTE(fanuc_style_start);
   1: XIC(fanuc_run)XIC(fanuc_permissive)[OTE(fanuc.uop.IMSTP) ,OTE(fanuc.uop.enable) ,OTE(fanuc.uop.SFSPD) ];
   2: GRT(fanuc.reg.target_boxnum,6)LES(fanuc.reg.target_boxnum,9)LES(fanuc.reg.target_slotrow,fanuc.reg.boxtype.numrows)LES(fanuc.reg.target_slotcol,fanuc.reg.boxtype.numcols)OTE(fanuc_target_valid);
END_ROUTINE

ROUTINE fanuc_IO   (* ladder *)
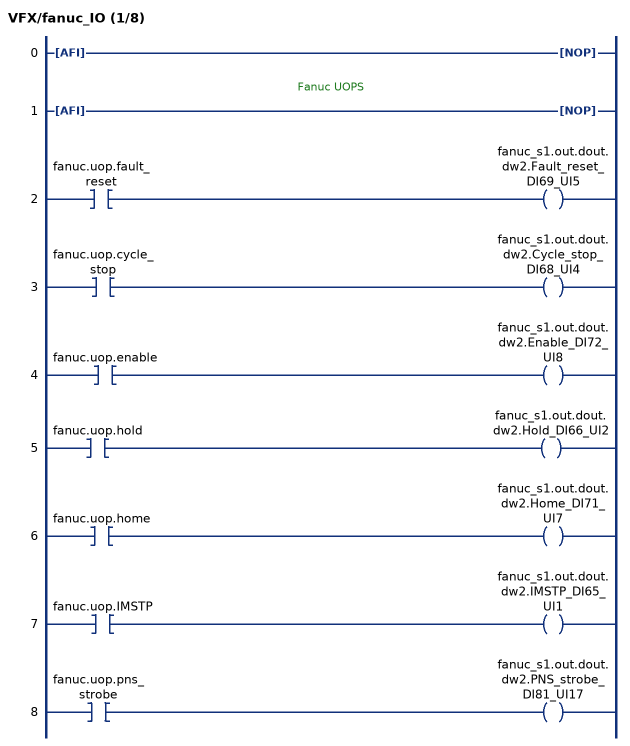
   0: AFI()NOP();
   // Fanuc UOPS
   1: AFI()NOP();
   2: XIC(fanuc.uop.fault_reset)OTE(fanuc_s1.out.dout.dw2.Fault_reset_DI69_UI5);
   3: XIC(fanuc.uop.cycle_stop)OTE(fanuc_s1.out.dout.dw2.Cycle_stop_DI68_UI4);
   4: XIC(fanuc.uop.enable)OTE(fanuc_s1.out.dout.dw2.Enable_DI72_UI8);
   5: XIC(fanuc.uop.hold)OTE(fanuc_s1.out.dout.dw2.Hold_DI66_UI2);
   6: XIC(fanuc.uop.home)OTE(fanuc_s1.out.dout.dw2.Home_DI71_UI7);
   7: XIC(fanuc.uop.IMSTP)OTE(fanuc_s1.out.dout.dw2.IMSTP_DI65_UI1);
   8: XIC(fanuc.uop.pns_strobe)OTE(fanuc_s1.out.dout.dw2.PNS_strobe_DI81_UI17);
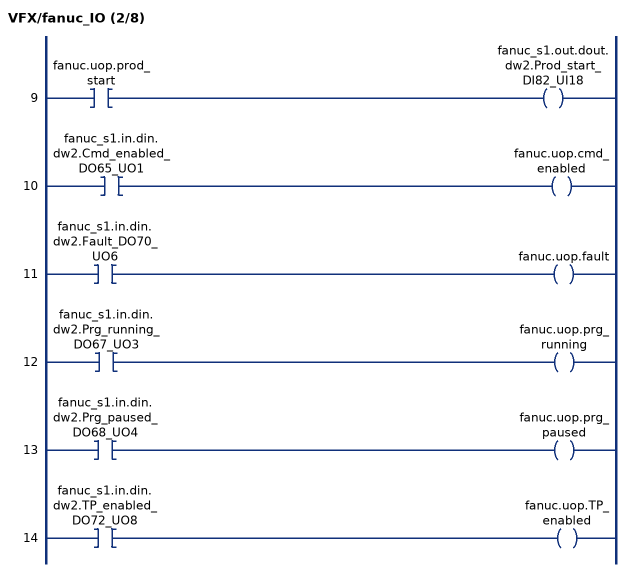
   9: XIC(fanuc.uop.prod_start)OTE(fanuc_s1.out.dout.dw2.Prod_start_DI82_UI18);
   10: XIC(fanuc_s1.in.din.dw2.Cmd_enabled_DO65_UO1)OTE(fanuc.uop.cmd_enabled);
   11: XIC(fanuc_s1.in.din.dw2.Fault_DO70_UO6)OTE(fanuc.uop.fault);
   12: XIC(fanuc_s1.in.din.dw2.Prg_running_DO67_UO3)OTE(fanuc.uop.prg_running);
   13: XIC(fanuc_s1.in.din.dw2.Prg_paused_DO68_UO4)OTE(fanuc.uop.prg_paused);
   14: XIC(fanuc_s1.in.din.dw2.TP_enabled_DO72_UO8)OTE(fanuc.uop.TP_enabled);
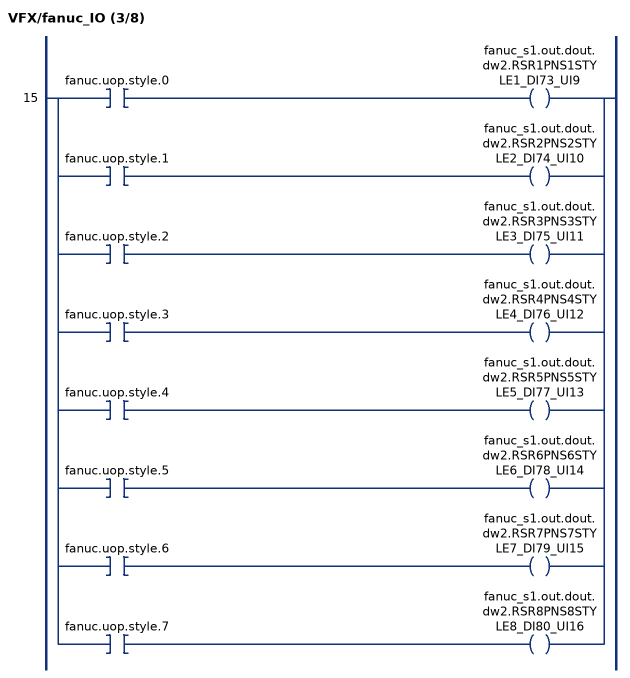
   15: [XIC(fanuc.uop.style.0) OTE(fanuc_s1.out.dout.dw2.RSR1PNS1STYLE1_DI73_UI9) ,XIC(fanuc.uop.style.1) OTE(fanuc_s1.out.dout.dw2.RSR2PNS2STYLE2_DI74_UI10) ,XIC(fanuc.uop.style.2) OTE(fanuc_s1.out.dout.dw2.RSR3PNS3STYLE3_DI75_UI11) ,XIC(fanuc.uop.style.3) OTE(fanuc_s1.out.dout.dw2.RSR4PNS4STYLE4_DI76_UI12) ,XIC(fanuc.uop.style.4) OTE(fanuc_s1.out.dout.dw2.RSR5PNS5STYLE5_DI77_UI13) ,XIC(fanuc.uop.style.5) OTE(fanuc_s1.out.dout.dw2.RSR6PNS6STYLE6_DI78_UI14) ,XIC(fanuc.uop.style.6) OTE(fanuc_s1.out.dout.dw2.RSR7PNS7STYLE7_DI79_UI15) ,XIC(fanuc.uop.style.7) OTE(fanuc_s1.out.dout.dw2.RSR8PNS8STYLE8_DI80_UI16) ];
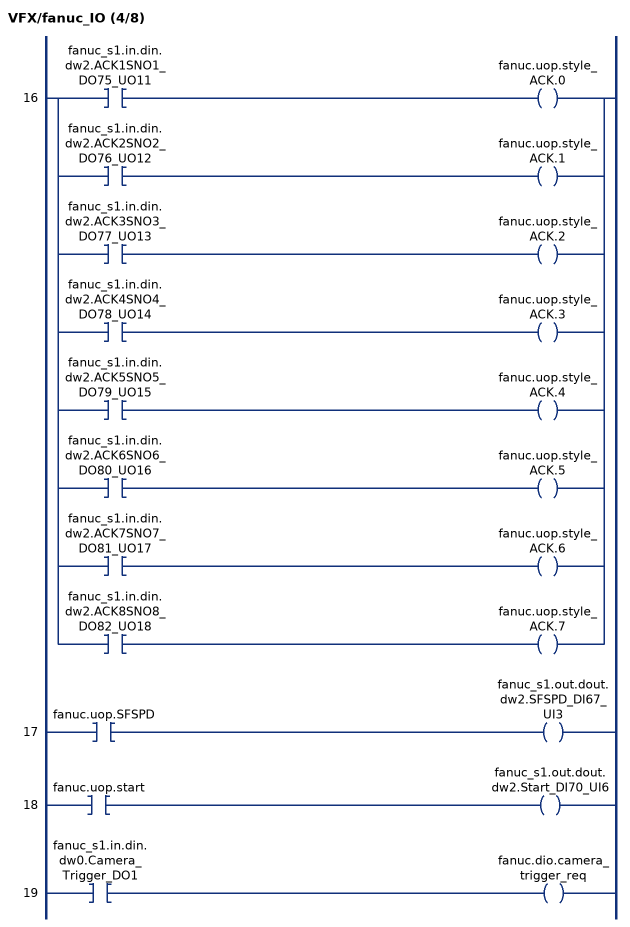
   16: [XIC(fanuc_s1.in.din.dw2.ACK1SNO1_DO75_UO11) OTE(fanuc.uop.style_ACK.0) ,XIC(fanuc_s1.in.din.dw2.ACK2SNO2_DO76_UO12) OTE(fanuc.uop.style_ACK.1) ,XIC(fanuc_s1.in.din.dw2.ACK3SNO3_DO77_UO13) OTE(fanuc.uop.style_ACK.2) ,XIC(fanuc_s1.in.din.dw2.ACK4SNO4_DO78_UO14) OTE(fanuc.uop.style_ACK.3) ,XIC(fanuc_s1.in.din.dw2.ACK5SNO5_DO79_UO15) OTE(fanuc.uop.style_ACK.4) ,XIC(fanuc_s1.in.din.dw2.ACK6SNO6_DO80_UO16) OTE(fanuc.uop.style_ACK.5) ,XIC(fanuc_s1.in.din.dw2.ACK7SNO7_DO81_UO17) OTE(fanuc.uop.style_ACK.6) ,XIC(fanuc_s1.in.din.dw2.ACK8SNO8_DO82_UO18) OTE(fanuc.uop.style_ACK.7) ];
   17: XIC(fanuc.uop.SFSPD)OTE(fanuc_s1.out.dout.dw2.SFSPD_DI67_UI3);
   18: XIC(fanuc.uop.start)OTE(fanuc_s1.out.dout.dw2.Start_DI70_UI6);
   19: XIC(fanuc_s1.in.din.dw0.Camera_Trigger_DO1)OTE(fanuc.dio.camera_trigger_req);
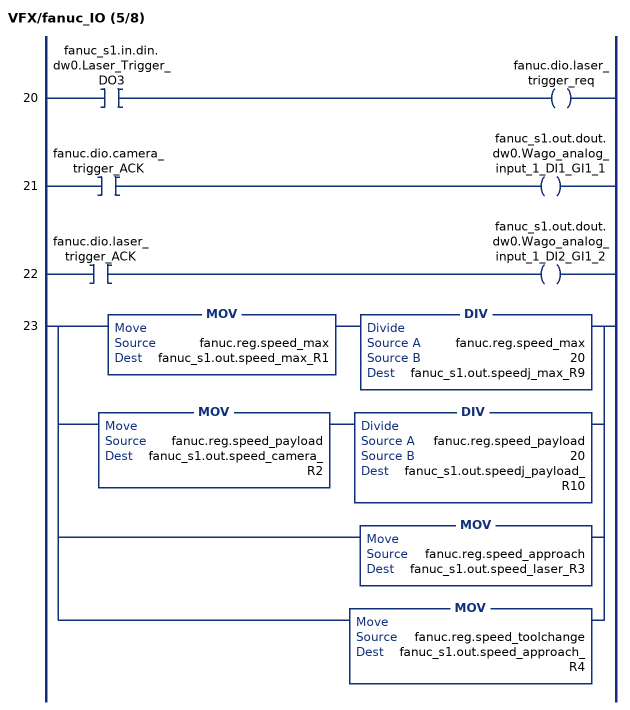
   20: XIC(fanuc_s1.in.din.dw0.Laser_Trigger_DO3)OTE(fanuc.dio.laser_trigger_req);
   21: XIC(fanuc.dio.camera_trigger_ACK)OTE(fanuc_s1.out.dout.dw0.Wago_analog_input_1_DI1_GI1_1);
   22: XIC(fanuc.dio.laser_trigger_ACK)OTE(fanuc_s1.out.dout.dw0.Wago_analog_input_1_DI2_GI1_2);
   23: [MOV(fanuc.reg.speed_max,fanuc_s1.out.speed_max_R1) DIV(fanuc.reg.speed_max,20,fanuc_s1.out.speedj_max_R9) ,MOV(fanuc.reg.speed_payload,fanuc_s1.out.speed_camera_R2) DIV(fanuc.reg.speed_payload,20,fanuc_s1.out.speedj_payload_R10) ,MOV(fanuc.reg.speed_approach,fanuc_s1.out.speed_laser_R3) ,MOV(fanuc.reg.speed_toolchange,fanuc_s1.out.speed_approach_R4) ];
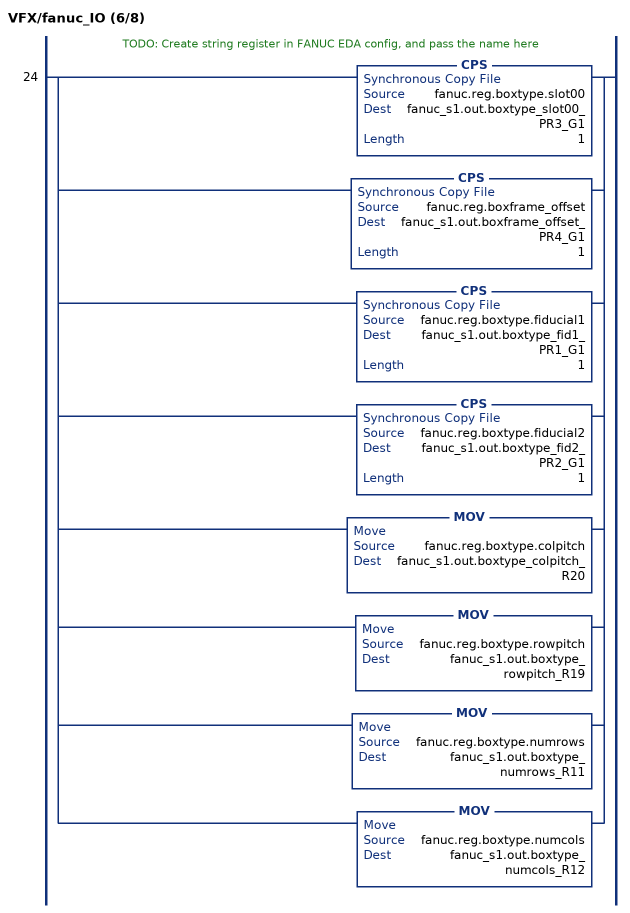
   // TODO: Create string register in FANUC EDA config, and pass the name here
   24: [CPS(fanuc.reg.boxtype.slot00,fanuc_s1.out.boxtype_slot00_PR3_G1,1) ,CPS(fanuc.reg.boxframe_offset,fanuc_s1.out.boxframe_offset_PR4_G1,1) ,CPS(fanuc.reg.boxtype.fiducial1,fanuc_s1.out.boxtype_fid1_PR1_G1,1) ,CPS(fanuc.reg.boxtype.fiducial2,fanuc_s1.out.boxtype_fid2_PR2_G1,1) ,MOV(fanuc.reg.boxtype.colpitch,fanuc_s1.out.boxtype_colpitch_R20) ,MOV(fanuc.reg.boxtype.rowpitch,fanuc_s1.out.boxtype_rowpitch_R19) ,MOV(fanuc.reg.boxtype.numrows,fanuc_s1.out.boxtype_numrows_R11) ,MOV(fanuc.reg.boxtype.numcols,fanuc_s1.out.boxtype_numcols_R12) ];
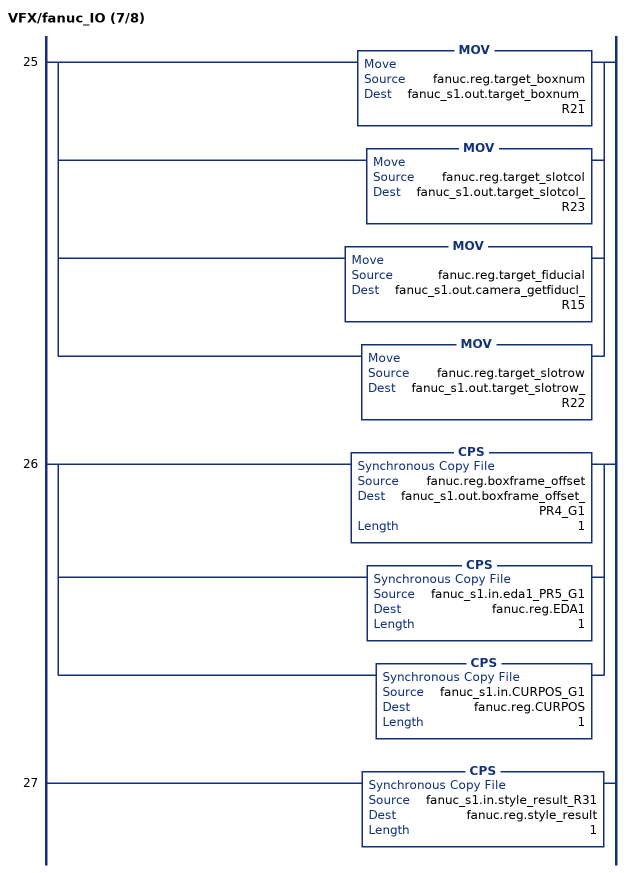
   25: [MOV(fanuc.reg.target_boxnum,fanuc_s1.out.target_boxnum_R21) ,MOV(fanuc.reg.target_slotcol,fanuc_s1.out.target_slotcol_R23) ,MOV(fanuc.reg.target_fiducial,fanuc_s1.out.camera_getfiducl_R15) ,MOV(fanuc.reg.target_slotrow,fanuc_s1.out.target_slotrow_R22) ];
   26: [CPS(fanuc.reg.boxframe_offset,fanuc_s1.out.boxframe_offset_PR4_G1,1) ,CPS(fanuc_s1.in.eda1_PR5_G1,fanuc.reg.EDA1,1) ,CPS(fanuc_s1.in.CURPOS_G1,fanuc.reg.CURPOS,1) ];
   27: CPS(fanuc_s1.in.style_result_R31,fanuc.reg.style_result,1);
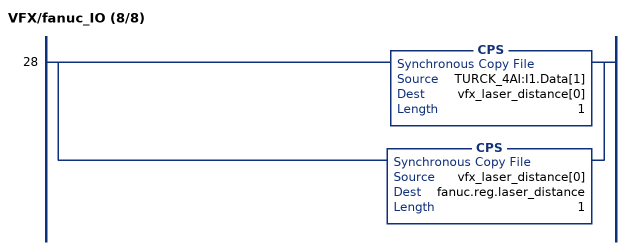
   28: [CPS(TURCK_4AI:I1.Data[1],vfx_laser_distance[0],1) ,CPS(vfx_laser_distance[0],fanuc.reg.laser_distance,1) ];
END_ROUTINE
